// TIA Portal V19 export
TYPE "LEXCHANGETRAY_typeRoller_toWorkStationRollerReq"
// stored: Access Published
   STRUCT
      inFeedReq : Bool;
      outFeedReq : Bool;   // 请求排料排料
   END_STRUCT;
END_TYPE
